{attribute 'qualified_only'}
TYPE E_TransportTube :
(
	LS1 := 0,
	LS5 := 1,
	LS8 := 2,
	LD2 := 3,
	LD4 := 4,
	LD6 := 5,
	LD8 := 6,
	LD9 := 7,
	LD10 := 8,
	LD14 := 9
) UINT;
END_TYPE

(* stored: Version 1.1.0.1, ProductVersion 3.1.4022.18
   DUT E_TransportTube: Id {26e13819-1baa-4350-8f0d-08839603bdb0} *)
